// TIA Portal V20 export
TYPE "LER_typeAlignCalibrationMonitoring"
// stored: Access Published
   STRUCT
      stepSequence : DInt;
      alignTableAxisXPosition : LReal;
      alignTableAxisY1Position : LReal;
      alignTableAxisY2Position : LReal;
      busy : Bool;
      error : Bool;
      done : Bool;
   END_STRUCT;
END_TYPE
